// TwinCAT 3 PLC project HOMS_Test_PLC
// ProgramVersion: 3.1.4020.5
// libraries:
//   lcls-twincat-motion, * (SLAC)
//   Tc2_MC2, * (Beckhoff Automation GmbH)
//   Tc2_Standard, * (Beckhoff Automation GmbH)
//   Tc2_System, * (Beckhoff Automation GmbH)
//   Tc2_Utilities, * (Beckhoff Automation GmbH)
//   Tc3_Module, * (Beckhoff Automation GmbH)
// project tree:
//   / PlcTask.TcTTO (not stored)
//   POUs/ Main.TcPOU
// real-time tasks:
//   TASK PlcTask: cycle T#10ms, priority 20, ADS port 350
// motion (NC):
//   TASK NC-Task 1 SAF: cycle T#2ms, priority 4, ADS port 501
//   TASK NC-Task 1 SVB: cycle T#10ms, priority 8, ADS port 511
//   AXIS Axis_Yup (id 3)
//     Dynamic: DelayTime=0.008
//     Velo: Maximum=0.45
//     OtherSettings: AllowMotionCmdToSlave=true
//     encoder EncType=1
//       EncPara: ScaleFactorNumerator=1e-06
//     drive DrvType=5
//       Analog: ScaleFactorActTorque=0.1
//       TimeComp: TaskDelayCycles=1
//     controller CtrType=2
//       CtrPara: PriorControlFactor=1
//         PosDiffControl: Range=1
//         Observer: BandWidth=20
//   AXIS Axis_Ydwn (id 4)
//     Dynamic: DelayTime=0.008
//     Velo: Maximum=0.45
//     OtherSettings: AllowMotionCmdToSlave=true
//     encoder EncType=1
//       EncPara: ScaleFactorNumerator=1e-06
//     drive DrvType=5
//       Analog: ScaleFactorActTorque=0.1
//       TimeComp: TaskDelayCycles=1
//     controller CtrType=2
//       CtrPara: PriorControlFactor=1
//         PosDiffControl: Range=1
//         Observer: BandWidth=20
//   AXIS Axis_Xup (id 1)
//     Dynamic: Acceleration=2, Deceleration=2, DelayTime=0.008
//     Velo: Maximum=1
//     OtherSettings: AllowMotionCmdToSlave=true
//     encoder EncType=1
//       EncPara: ScaleFactorNumerator=1e-06
//     drive DrvType=5
//       Analog: VeloReferenz=1.2206875, ScaleFactorActTorque=0.1
//       TimeComp: TaskDelayCycles=1
//     controller CtrType=2
//       CtrPara: PriorControlFactor=1
//         PosDiffControl: Range=1
//         PID: PosKp=10, PosExtKp=1, DeadBandPosition=4e-05
//         Observer: BandWidth=20
//   AXIS Axis_Xdwn (id 2)
//     Dynamic: Acceleration=2, Deceleration=2, DelayTime=0.008
//     Velo: Maximum=1
//     OtherSettings: AllowMotionCmdToSlave=true
//     encoder EncType=1
//       EncPara: ScaleFactorNumerator=1e-06
//     drive DrvType=5
//       Analog: VeloReferenz=1.2206875, ScaleFactorActTorque=0.1
//       TimeComp: TaskDelayCycles=1
//     controller CtrType=2
//       CtrPara: PriorControlFactor=1
//         PosDiffControl: Range=1
//         PID: PosKp=10, PosExtKp=1, DeadBandPosition=4e-05
//         Observer: BandWidth=20
//   AXIS Axis_PitchCoarse (id 5)
//     Dynamic: Acceleration=0.5, Deceleration=0.5, DelayTime=0.008
//     Velo: Maximum=0.3
//     OtherSettings: AllowMotionCmdToSlave=true
//     encoder EncType=1
//       EncPara: ScaleFactorNumerator=1e-006
//     drive DrvType=5
//       Analog: VeloReferenz=0.39062, ScaleFactorActTorque=0.1
//       TimeComp: TaskDelayCycles=1
//     controller CtrType=2
//       CtrPara: PriorControlFactor=1
//         PosDiffControl: Range=0.0006
//         PID: PosKp=10, PosExtKp=1, DeadBandPosition=4e-005
//         Observer: BandWidth=20
//   AXIS Axis_Bender (id 6)
// variable links:
//   HOMS_Test_PLC Instance <-> NC-Task 1 SAF/Axes/Axis_Bender
//     PlcTask Inputs/Main.M6.Axis.NcToPlc <-> Outputs/ToPlc
//     PlcTask Outputs/Main.M6.Axis.PlcToNc <-> Inputs/FromPlc
//   HOMS_Test_PLC Instance <-> NC-Task 1 SAF/Axes/Axis_PitchCoarse
//     PlcTask Inputs/Main.M5.Axis.NcToPlc <-> Outputs/ToPlc
//     PlcTask Outputs/Main.M5.Axis.PlcToNc <-> Inputs/FromPlc
//   HOMS_Test_PLC Instance <-> NC-Task 1 SAF/Axes/Axis_Xdwn
//     PlcTask Inputs/Main.M2.Axis.NcToPlc <-> Outputs/ToPlc
//     PlcTask Outputs/Main.M2.Axis.PlcToNc <-> Inputs/FromPlc
//   HOMS_Test_PLC Instance <-> NC-Task 1 SAF/Axes/Axis_Xup
//     PlcTask Inputs/Main.M1.Axis.NcToPlc <-> Outputs/ToPlc
//     PlcTask Outputs/Main.M1.Axis.PlcToNc <-> Inputs/FromPlc
//   HOMS_Test_PLC Instance <-> NC-Task 1 SAF/Axes/Axis_Ydwn
//     PlcTask Inputs/Main.M4.Axis.NcToPlc <-> Outputs/ToPlc
//     PlcTask Outputs/Main.M4.Axis.PlcToNc <-> Inputs/FromPlc
//   HOMS_Test_PLC Instance <-> NC-Task 1 SAF/Axes/Axis_Yup
//     PlcTask Inputs/Main.M3.Axis.NcToPlc <-> Outputs/ToPlc
//     PlcTask Outputs/Main.M3.Axis.PlcToNc <-> Inputs/FromPlc

// ---- POUs/Main.TcPOU
PROGRAM Main
VAR
    M3: DUT_MotionStage; // Yup
	{attribute 'pytmc' := '
	  pv: AXISYUP
	'}
	fbMotionStage_y_up : FB_MotionStage;

	M4: DUT_MotionStage; // Ydwn
	{attribute 'pytmc' := '
	  pv: AXISYDWN
	'}
	fbMotionStage_y_dwn : FB_MotionStage;

	M1: DUT_MotionStage:=(nCommand:=3); // Xup
	{attribute 'pytmc' := '
	  pv: AXISXUP
	'}
	fbMotionStage_x_up : FB_MotionStage;

	M2: DUT_MotionStage:=(nCommand:=3); // Xdwn
	{attribute 'pytmc' := '
	  pv: AXISXDWN
	'}
	fbMotionStage_x_dwn : FB_MotionStage;

	M5: DUT_MotionStage:=(nCommand:=3); // PitchCoarse
	{attribute 'pytmc' := '
	  pv: AXISPITCH
	'}
	fbMotionStage_pitch : FB_MotionStage;

	M6: DUT_MotionStage:=(nCommand:=3); // Bender
	{attribute 'pytmc' := '
	  pv: AXISBENDER
	'}
	fbMotionStage_bender : FB_MotionStage;

	{attribute 'pytmc' := '
	  pv: TEST:MAIN:STOENABLE
	  io: io
	'}
	stoEnable AT %I* : BOOL;

	x_up_enc  AT %I*: ST_RenishawAbsEnc;
	x_dwn_enc  AT %I*: ST_RenishawAbsEnc;	
	y_up_enc  AT %I*: ST_RenishawAbsEnc;
	y_dwn_enc  AT %I*: ST_RenishawAbsEnc:=(Ref:=0);

	// Auto coupling function block
	fbAutoCoupleX : FB_GantryAutoCoupling;
	fbAutoCoupleY : FB_GantryAutoCoupling;

	bExecuteCoupleX : BOOL;
	bExecuteCoupleY : BOOL;
	bExecuteDecoupleX : BOOL;
	bExecuteDecoupleY : BOOL;
	bGantryAlreadyCoupledX : BOOL;
	bGantryAlreadyCoupledY : BOOL;
	
	// Gantry variables
//	fEncFudgeFactor : REAL := 1.005;
	nCurrGantryX : LINT;
	nCurrGantryY : LINT;
	nGantryTolX : LINT := 25000;
	nGantryTolY : LINT := 25000;
END_VAR

M1.bLimitForwardEnable := TRUE;
M1.bLimitBackwardEnable := TRUE;
M1.bPowerSelf := TRUE;
M1.nEnableMode := ENUM_StageEnableMode.STAGE_ENABLE_ALWAYS;

M2.bLimitForwardEnable := TRUE;
M2.bLimitBackwardEnable := TRUE;
M2.bPowerSelf := TRUE;
M2.nEnableMode := ENUM_StageEnableMode.STAGE_ENABLE_ALWAYS;

M3.bLimitForwardEnable := TRUE;
M3.bLimitBackwardEnable := TRUE;
M3.bPowerSelf := TRUE;
M3.nEnableMode := ENUM_StageEnableMode.STAGE_ENABLE_ALWAYS;

M4.bLimitForwardEnable := TRUE;
M4.bLimitBackwardEnable := TRUE;
M4.bPowerSelf := TRUE;
M4.nEnableMode := ENUM_StageEnableMode.STAGE_ENABLE_ALWAYS;

M5.bLimitForwardEnable := TRUE;
M5.bLimitBackwardEnable := TRUE;
M5.bPowerSelf := TRUE;
M5.nEnableMode := ENUM_StageEnableMode.STAGE_ENABLE_ALWAYS;

M6.bLimitForwardEnable := TRUE;
M6.bLimitBackwardEnable := TRUE;
M6.bPowerSelf := TRUE;
M6.nEnableMode := ENUM_StageEnableMode.STAGE_ENABLE_ALWAYS;

// Buttons to enable motors: write 0 to enable, 2 to disable
//M1.nEnableMode; // Yup
//M2.nEnableMode; // Ydwn
//M3.nEnableMode; // Xup
//M4.nEnableMode; // Xdwn
//M5.nEnableMode; // PitchCoarse
//M6.nEnableMode; // Bender

// Encoder Reference Values:
y_up_enc.Ref := 0;
y_dwn_enc.Ref := 0;
x_up_enc.Ref := 0; 
x_dwn_enc.Ref := 0;

// Pretend encoder counts
//y_up_enc.Count := LREAL_TO_ULINT(M1.stAxisStatus.fActPosition * fEncFudgeFactor * EXPT(10, 6));
//y_dwn_enc.Count := LREAL_TO_ULINT(M2.stAxisStatus.fActPosition * EXPT(10, 6));

//x_up_enc.Count := LREAL_TO_ULINT(M3.stAxisStatus.fActPosition * fEncFudgeFactor * EXPT(10, 6));
//x_dwn_enc.Count := LREAL_TO_ULINT(M4.stAxisStatus.fActPosition * EXPT(10, 6));

// Gantry Differences to monitor
//nCurrGantryY := ((ULINT_TO_LINT(y_up_enc.Count) - ULINT_TO_LINT(y_up_enc.Ref)) - (ULINT_TO_LINT(y_dwn_enc.Count) - ULINT_TO_LINT(y_dwn_enc.Ref)));
//nCurrGantryX := ((ULINT_TO_LINT(x_up_enc.Count) - ULINT_TO_LINT(x_up_enc.Ref)) - (ULINT_TO_LINT(x_dwn_enc.Count) - ULINT_TO_LINT(x_dwn_enc.Ref)));

//E-Stop
M1.bHardwareEnable := stoEnable;
M2.bHardwareEnable := stoEnable;
M3.bHardwareEnable := stoEnable;
M4.bHardwareEnable := stoEnable;
M5.bHardwareEnable := stoEnable;
M6.bHardwareEnable := stoEnable;

// Start Autocoupling
fbAutoCoupleX(nGantryTol:=nGantryTolX, Master:=M1, MasterEnc:=x_up_enc, Slave:=M2,
	          SlaveEnc:=x_dwn_enc, bExecuteCouple:=bExecuteCoupleX,
              bExecuteDecouple:=bExecuteDecoupleX,
              bGantryAlreadyCoupled=>bGantryAlreadyCoupledX);

fbAutoCoupleY(nGantryTol:=nGantryTolY, Master:=M3, MasterEnc:=y_up_enc, Slave:=M4,
	          SlaveEnc:=y_dwn_enc, bExecuteCouple:=bExecuteCoupleY,
              bExecuteDecouple:=bExecuteDecoupleY,
			  bGantryAlreadyCoupled=>bGantryAlreadyCoupledY);

fbMotionStage_y_up  (stMotionStage:=M3);
fbMotionStage_y_dwn (stMotionStage:=M4);
fbMotionStage_x_up  (stMotionStage:=M1);
fbMotionStage_x_dwn (stMotionStage:=M2);
fbMotionStage_pitch (stMotionStage:=M5);
fbMotionStage_bender (stMotionStage:=M6);

END_PROGRAM
